// TIA Portal V20 export
TYPE "zd_SCS_ModeBox_Inputs"
// stored: Access Published, IsFailsafeCompliant true, Namespace Safety
   STRUCT
      SI1_Setup : Bool;   // SAFE INPUT 1 SETUP
      SI2_Auto : Bool;   // SAFE INPUT 2 AUTO
      SI3_Disable : Bool;   // SAFE INPUT 3 DISABLE
   END_STRUCT;
END_TYPE
